Universal Robots PolyScope program: orange_Wheel_holder.urp

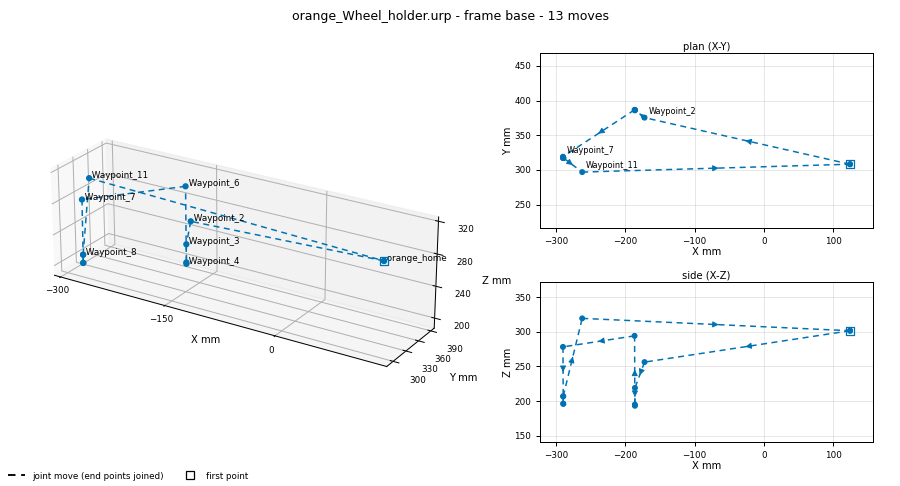
[picture p0: tool path of orange_Wheel_holder.urp in frame base, 13 of 13 moves have a stored position in this frame; points joined in program order, loops and branches not executed]
Program orange_Wheel_holder (installation=default directory=/programs/usbdisk/Zahra1/orangi createdIn=5.11.11.1010533 lastSavedIn=5.11.11.1010533 robotSerialNumber=20205300864)
Calibrated DH parameters: a=[-0.000166, -0.243494, -0.153108, 0.000057, -0.000123, 0]; d=[0.151897, -1.34267, 53.988124, -52.514559, 0.085283, 0.092193]; alpha=[1.572472, -0.003756, 0.002824, 1.570807, -1.572621, 0]; deltaTheta=[0, 0.020704, 7.033215, -0.770746, 0.000004, 0]
Robot Program (runOnlyOnce=true)
  MoveJ speed 60 deg/s, acceleration 80 deg/s^2 (useActiveTCP=true) feature=Base
    Waypoint orange_home: TCP in base x=124.286 y=308.277 z=301.462 mm, rx=2.2499 ry=-2.1846 rz=-0.0963 rad; joints [-269.66, -91.226, -90.279, -86.086, 92.69, 808.818] deg
    Waypoint Waypoint_2: TCP in base x=-172.055 y=375.417 z=256.216 mm, rx=-3.0657 ry=0.0098 rz=0.0647 rad; joints [-226.696, -111.293, -78.961, -74.855, 88.746, 763.729] deg
    URCap Gripper (Robotiq_Grippers, Robotiq Inc.) dataModel(position=25.098039215686274, force=94.0, speed=40.0, positionInDouble=25.098039215686274, forceInDouble=94.0, speedInDouble=40.0, slaveIds=[9], blocking=true, robotCompliant=false)
    Waypoint Waypoint_3: TCP in base x=-185.901 y=386.345 z=219.02 mm, rx=3.129 ry=-0.0067 rz=0.0147 rad; joints [-226.635, -118.916, -75.362, -76.507, 90.049, 763.722] deg
    Waypoint Waypoint_4: TCP in base x=-185.931 y=386.144 z=193.243 mm, rx=3.1315 ry=-0.0059 rz=0.0136 rad; joints [-226.607, -120.689, -79.846, -70.12, 89.98, 763.73] deg
    URCap Gripper (Robotiq_Grippers, Robotiq Inc.) dataModel(position=75.68627450980392, force=94.0, speed=40.0, positionInDouble=75.68627450980392, forceInDouble=94.0, speedInDouble=40.0, slaveIds=[9], blocking=true, robotCompliant=false)
    Waypoint Waypoint_5: TCP in base x=-186.008 y=386.092 z=195.041 mm, rx=3.1348 ry=-0.0059 rz=0.0063 rad; joints [-226.609, -120.467, -79.825, -70.044, 90.048, 763.73] deg
    Waypoint Waypoint_6: TCP in base x=-186.417 y=386.759 z=294.08 mm, rx=3.1348 ry=-0.0059 rz=0.0064 rad; joints [-226.582, -117.349, -57.627, -95.363, 90.013, 763.704] deg
    Waypoint Waypoint_7: TCP in base x=-289.696 y=319.124 z=278.159 mm, rx=3.1045 ry=-0.0856 rz=0.0905 rad; joints [-210.168, -119.21, -57.721, -96.844, 90.059, 783.062] deg
    Waypoint Waypoint_8: TCP in base x=-289.354 y=317.472 z=206.884 mm, rx=3.1089 ry=-0.0204 rz=0.0128 rad; joints [-210.311, -120.184, -76.561, -74.488, 91.33, 780.542] deg
    Waypoint Waypoint_9: TCP in base x=-289.272 y=317.131 z=196.151 mm, rx=3.1089 ry=-0.0204 rz=0.0127 rad; joints [-210.28, -120.91, -78.424, -71.896, 91.331, 780.578] deg
    URCap Gripper (Robotiq_Grippers, Robotiq Inc.) dataModel(position=25.098039215686274, force=94.0, speed=40.0, positionInDouble=25.098039215686274, forceInDouble=94.0, speedInDouble=40.0, slaveIds=[9], blocking=true, robotCompliant=false)
    Waypoint Waypoint_9: TCP in base x=-289.272 y=317.131 z=196.151 mm, rx=3.1089 ry=-0.0204 rz=0.0127 rad; joints [-210.28, -120.91, -78.424, -71.896, 91.331, 780.578] deg
    Waypoint Waypoint_8: TCP in base x=-289.354 y=317.472 z=206.884 mm, rx=3.1089 ry=-0.0204 rz=0.0128 rad; joints [-210.311, -120.184, -76.561, -74.488, 91.33, 780.542] deg
    Waypoint Waypoint_11: TCP in base x=-261.966 y=296.956 z=319.299 mm, rx=-3.0415 ry=0.0454 rz=0.0955 rad; joints [-208.521, -105.464, -70.368, -88.263, 86.635, 783.098] deg
    Waypoint orange_home: TCP in base x=124.286 y=308.277 z=301.462 mm, rx=2.2499 ry=-2.1846 rz=-0.0963 rad; joints [-269.66, -91.226, -90.279, -86.086, 92.69, 808.818] deg
